TYPE SDT :
STRUCT
	YEAR : INT;
	MONTH : INT;
	DAY : INT;
	WEEKDAY : INT;
	HOUR : INT;
	MINUTE : INT;
	SECOND : INT;
	MS : INT;
END_STRUCT
END_TYPE

(* stored: Version 1.1.0.1
   DUT SDT: Id {a7f09b4c-caeb-4613-87e8-e06f9203fc9d} *)
